{attribute 'enable_dynamic_creation'} 
FUNCTION_BLOCK FB_CustomShape IMPLEMENTS I_Shape
VAR_INPUT
END_VAR
VAR_OUTPUT
END_VAR
VAR
END_VAR

{warning 'Agregar implementación de método'}
METHOD M_Draw : BOOL
ADSLOGSTR(ADSLOG_MSGTYPE_HINT, 'Draw custom shape', '');
M_Draw := TRUE;
END_METHOD

END_FUNCTION_BLOCK

(* stored: Version 1.1.0.1, ProductVersion 3.1.4024.12
   POU FB_CustomShape: Id {15f198ef-d7e5-4b39-ba33-155e75a80fa1}, SpecialFunc None
   Method M_Draw: Id {162a5a28-7a78-4f3d-8f00-c95d475f840e} *)
